// TIA Portal V16 export
// export: Created 2024-09-05T17:40:13.8284058Z, ExportSetting WithDefaults, DisplayName Totally Integrated Automation Portal, DisplayVersion V16 Update 6, DisplayName TIA Portal Version Control Interface, DisplayVersion V16 Update 2, DisplayName TIA Portal Openness, DisplayVersion V16 Update 6, DisplayName STEP 7 Professional, DisplayVersion V16 Update 6, DisplayName STEP 7 Safety, DisplayVersion V16, DisplayName WinCC Advanced, DisplayVersion V16 Update 6
TYPE "UDT_Digiforce_send"
// stored: IsFailsafeCompliant false
   STRUCT
      Tare_X : Bool;
      Res_Stat : Bool;
      Stest : Bool;
      Strobe : Bool;
      Auto : Bool;
      reserve1 : Bool;
      reserve2 : Bool;
      reserve3 : Bool;
      Prog : Byte;
      Start : Bool;
   END_STRUCT;
END_TYPE
